(* Logix 5000 project; controller SX_V040001_C001 vendor 1 type 14 code 77 rev 16.23; software revision 16.04; part 20 of 35 *)
(* tags used below, declared in another part *)
   ALL_KINDS : INT[90];
   G_DInput : DINT[3];
   G_DOutput : DINT[3];
   METERING : INT[44];
   NOTDOS : INT[6];
   PARAMETER : INT[501];
(* MainProgram, continued *)

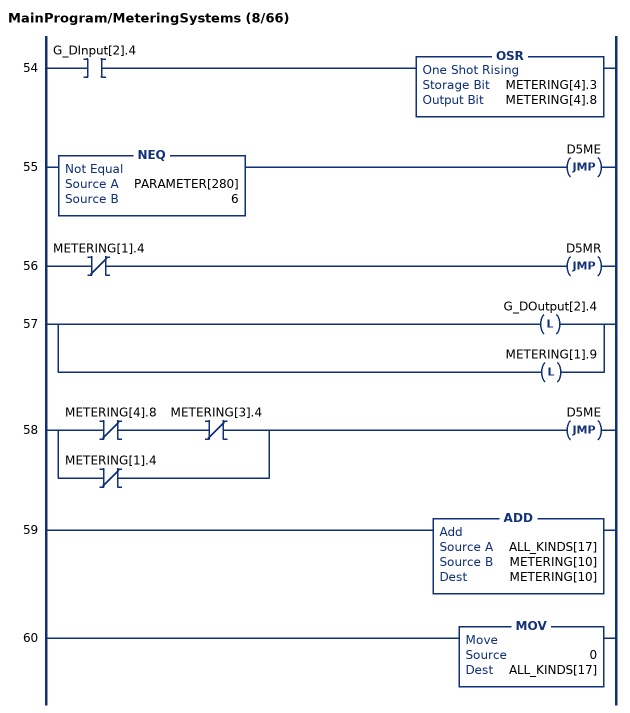
   [picture p432: MainProgram/MeteringSystems rungs 54-60]
   54: XIC(G_DInput[2].4)OSR(METERING[4].3,METERING[4].8);
   55: NEQ(PARAMETER[280],6)JMP(D5ME);
   56: XIO(METERING[1].4)JMP(D5MR);
   57: [OTL(G_DOutput[2].4) ,OTL(METERING[1].9) ];
   58: [XIO(METERING[4].8) XIO(METERING[3].4) ,XIO(METERING[1].4) ]JMP(D5ME);
   59: ADD(ALL_KINDS[17],METERING[10],METERING[10]);
   60: MOV(0,ALL_KINDS[17]);
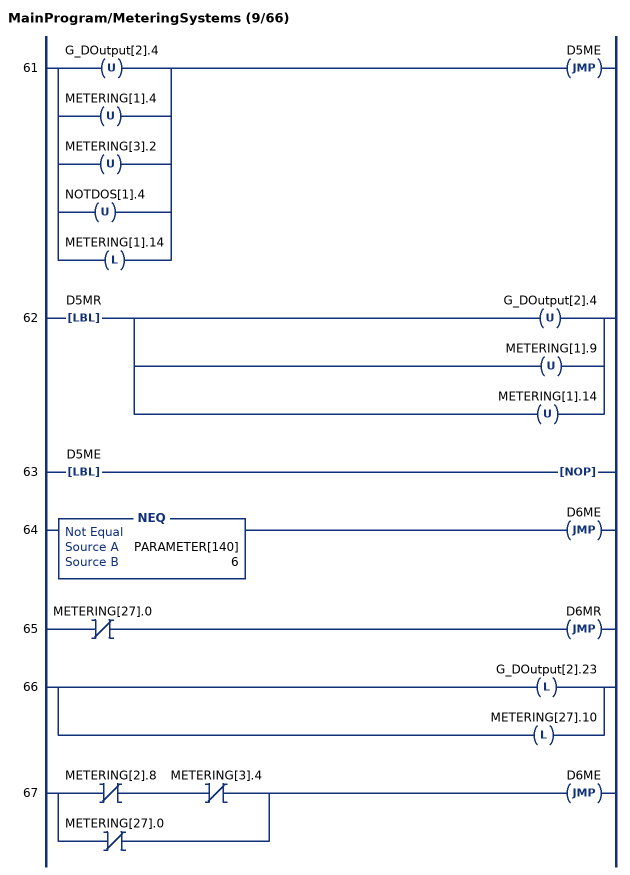
   61: [OTU(G_DOutput[2].4) ,OTU(METERING[1].4) ,OTU(METERING[3].2) ,OTU(NOTDOS[1].4) ,OTL(METERING[1].14) ]JMP(D5ME);
   62: LBL(D5MR)[OTU(G_DOutput[2].4) ,OTU(METERING[1].9) ,OTU(METERING[1].14) ];
   63: LBL(D5ME)NOP();
   64: NEQ(PARAMETER[140],6)JMP(D6ME);
   65: XIO(METERING[27].0)JMP(D6MR);
   66: [OTL(G_DOutput[2].23) ,OTL(METERING[27].10) ];
   67: [XIO(METERING[2].8) XIO(METERING[3].4) ,XIO(METERING[27].0) ]JMP(D6ME);
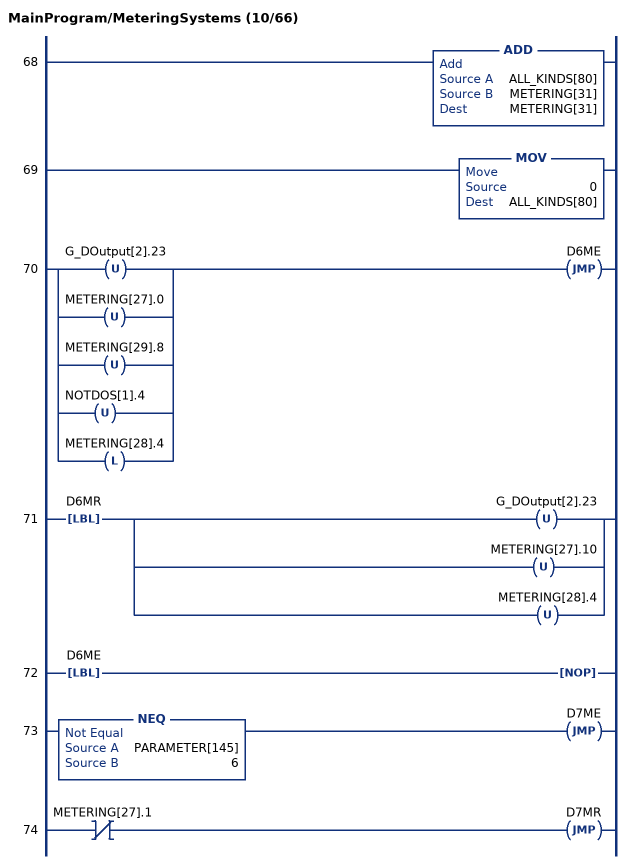
   68: ADD(ALL_KINDS[80],METERING[31],METERING[31]);
   69: MOV(0,ALL_KINDS[80]);
   70: [OTU(G_DOutput[2].23) ,OTU(METERING[27].0) ,OTU(METERING[29].8) ,OTU(NOTDOS[1].4) ,OTL(METERING[28].4) ]JMP(D6ME);
   71: LBL(D6MR)[OTU(G_DOutput[2].23) ,OTU(METERING[27].10) ,OTU(METERING[28].4) ];
   72: LBL(D6ME)NOP();
   73: NEQ(PARAMETER[145],6)JMP(D7ME);
   74: XIO(METERING[27].1)JMP(D7MR);
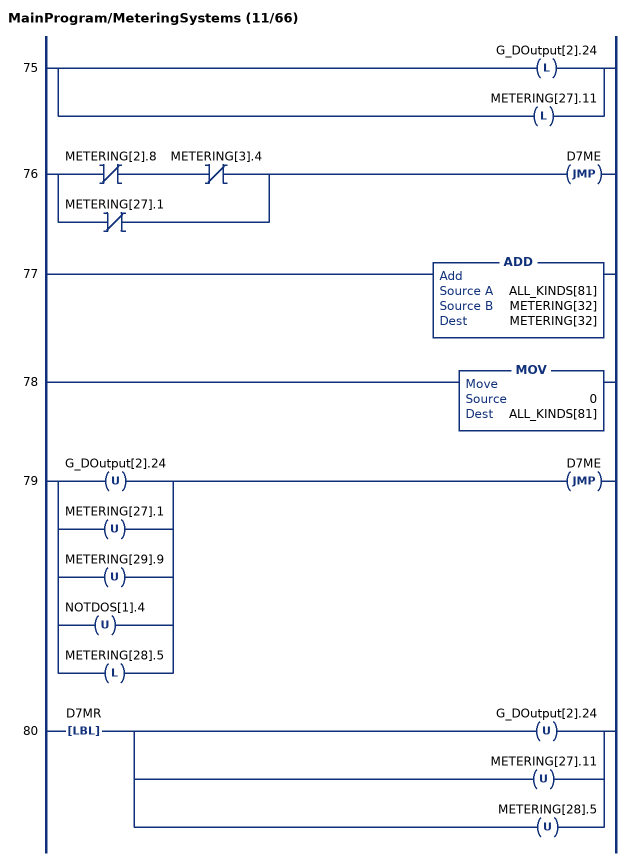
   75: [OTL(G_DOutput[2].24) ,OTL(METERING[27].11) ];
   76: [XIO(METERING[2].8) XIO(METERING[3].4) ,XIO(METERING[27].1) ]JMP(D7ME);
   77: ADD(ALL_KINDS[81],METERING[32],METERING[32]);
   78: MOV(0,ALL_KINDS[81]);
   79: [OTU(G_DOutput[2].24) ,OTU(METERING[27].1) ,OTU(METERING[29].9) ,OTU(NOTDOS[1].4) ,OTL(METERING[28].5) ]JMP(D7ME);
   80: LBL(D7MR)[OTU(G_DOutput[2].24) ,OTU(METERING[27].11) ,OTU(METERING[28].5) ];
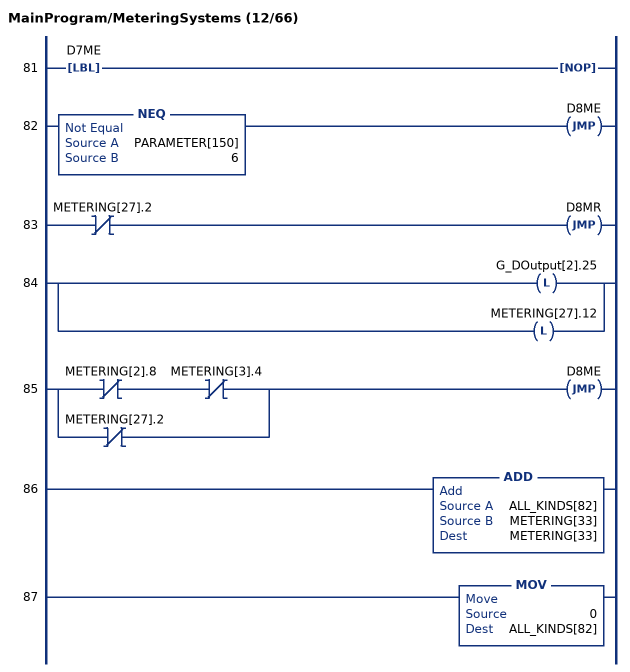
   81: LBL(D7ME)NOP();
   82: NEQ(PARAMETER[150],6)JMP(D8ME);
   83: XIO(METERING[27].2)JMP(D8MR);
   84: [OTL(G_DOutput[2].25) ,OTL(METERING[27].12) ];
   85: [XIO(METERING[2].8) XIO(METERING[3].4) ,XIO(METERING[27].2) ]JMP(D8ME);
   86: ADD(ALL_KINDS[82],METERING[33],METERING[33]);
   87: MOV(0,ALL_KINDS[82]);
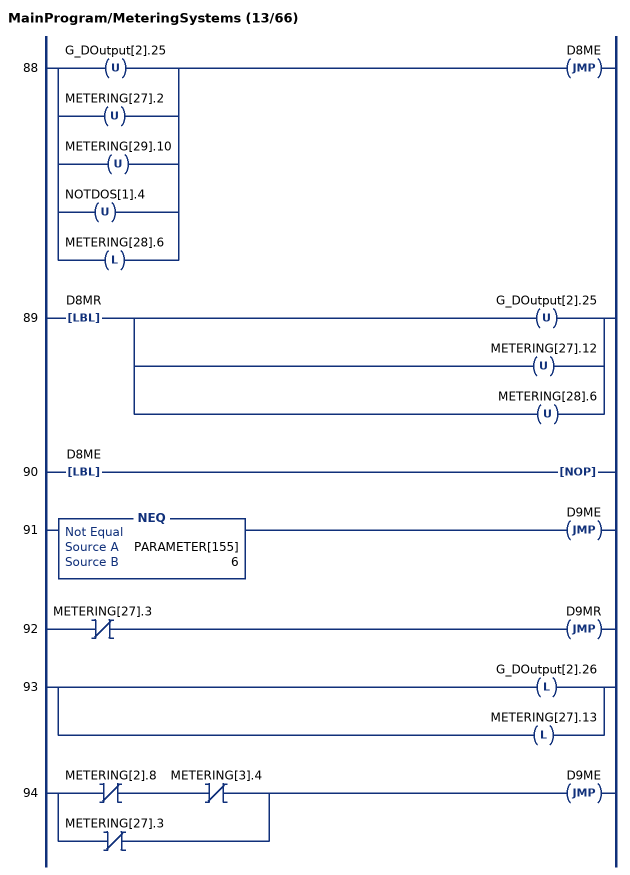
   88: [OTU(G_DOutput[2].25) ,OTU(METERING[27].2) ,OTU(METERING[29].10) ,OTU(NOTDOS[1].4) ,OTL(METERING[28].6) ]JMP(D8ME);
   89: LBL(D8MR)[OTU(G_DOutput[2].25) ,OTU(METERING[27].12) ,OTU(METERING[28].6) ];
   90: LBL(D8ME)NOP();
   91: NEQ(PARAMETER[155],6)JMP(D9ME);
   92: XIO(METERING[27].3)JMP(D9MR);
   93: [OTL(G_DOutput[2].26) ,OTL(METERING[27].13) ];
   94: [XIO(METERING[2].8) XIO(METERING[3].4) ,XIO(METERING[27].3) ]JMP(D9ME);
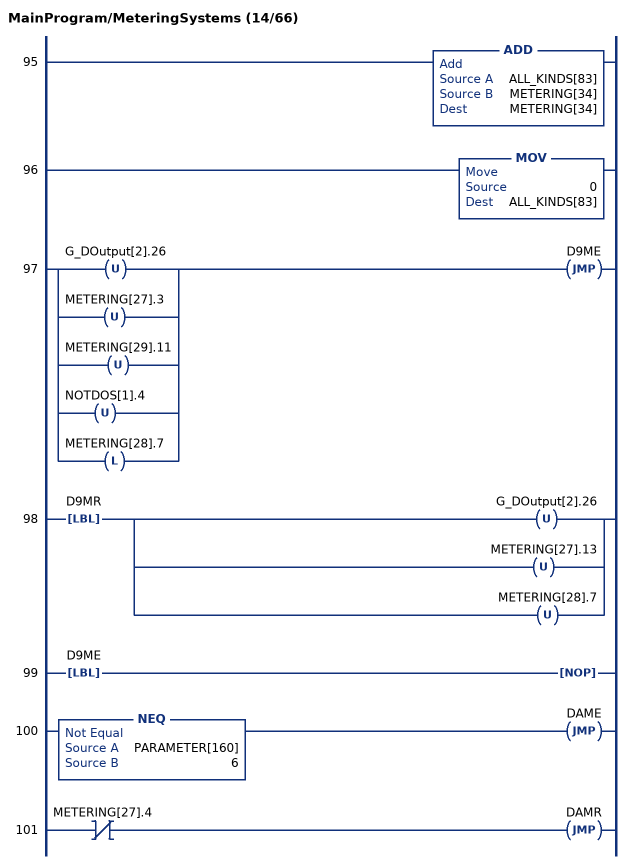
   95: ADD(ALL_KINDS[83],METERING[34],METERING[34]);
   96: MOV(0,ALL_KINDS[83]);
   97: [OTU(G_DOutput[2].26) ,OTU(METERING[27].3) ,OTU(METERING[29].11) ,OTU(NOTDOS[1].4) ,OTL(METERING[28].7) ]JMP(D9ME);
   98: LBL(D9MR)[OTU(G_DOutput[2].26) ,OTU(METERING[27].13) ,OTU(METERING[28].7) ];
   99: LBL(D9ME)NOP();
   100: NEQ(PARAMETER[160],6)JMP(DAME);
   101: XIO(METERING[27].4)JMP(DAMR);
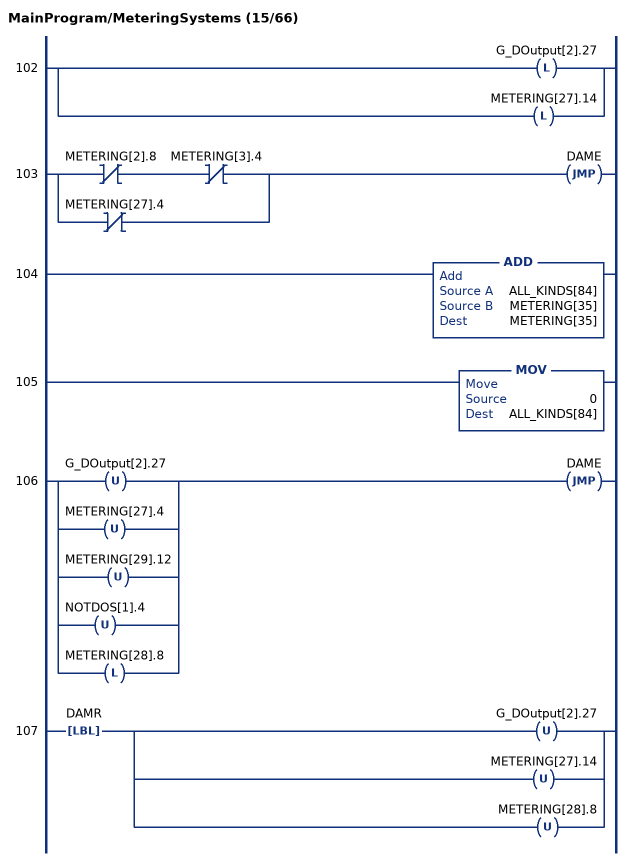
   102: [OTL(G_DOutput[2].27) ,OTL(METERING[27].14) ];
   103: [XIO(METERING[2].8) XIO(METERING[3].4) ,XIO(METERING[27].4) ]JMP(DAME);
   104: ADD(ALL_KINDS[84],METERING[35],METERING[35]);
   105: MOV(0,ALL_KINDS[84]);
   106: [OTU(G_DOutput[2].27) ,OTU(METERING[27].4) ,OTU(METERING[29].12) ,OTU(NOTDOS[1].4) ,OTL(METERING[28].8) ]JMP(DAME);
   107: LBL(DAMR)[OTU(G_DOutput[2].27) ,OTU(METERING[27].14) ,OTU(METERING[28].8) ];
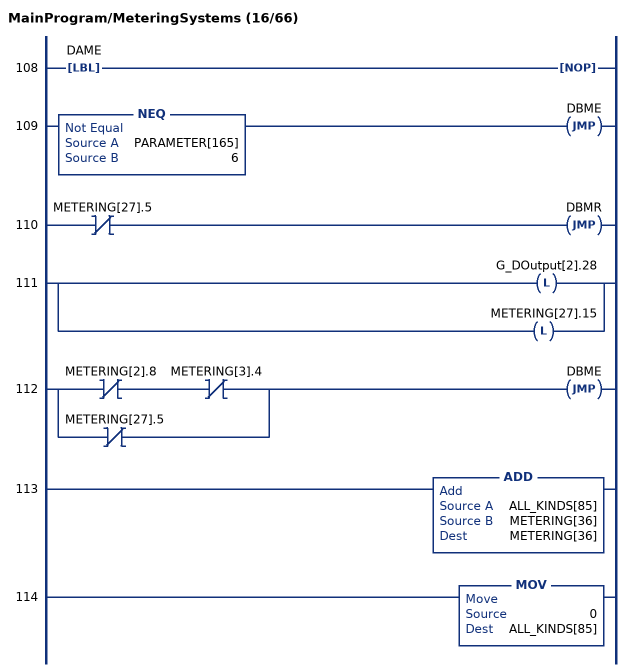
   108: LBL(DAME)NOP();
   109: NEQ(PARAMETER[165],6)JMP(DBME);
   110: XIO(METERING[27].5)JMP(DBMR);
   111: [OTL(G_DOutput[2].28) ,OTL(METERING[27].15) ];
   112: [XIO(METERING[2].8) XIO(METERING[3].4) ,XIO(METERING[27].5) ]JMP(DBME);
   113: ADD(ALL_KINDS[85],METERING[36],METERING[36]);
   114: MOV(0,ALL_KINDS[85]);
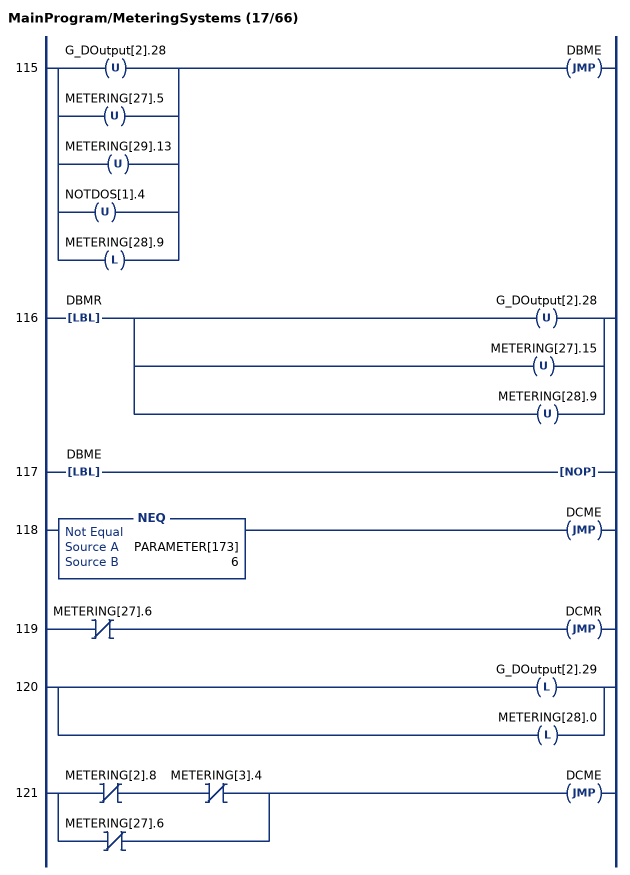
   115: [OTU(G_DOutput[2].28) ,OTU(METERING[27].5) ,OTU(METERING[29].13) ,OTU(NOTDOS[1].4) ,OTL(METERING[28].9) ]JMP(DBME);
   116: LBL(DBMR)[OTU(G_DOutput[2].28) ,OTU(METERING[27].15) ,OTU(METERING[28].9) ];
   117: LBL(DBME)NOP();
   118: NEQ(PARAMETER[173],6)JMP(DCME);
   119: XIO(METERING[27].6)JMP(DCMR);
   120: [OTL(G_DOutput[2].29) ,OTL(METERING[28].0) ];
   121: [XIO(METERING[2].8) XIO(METERING[3].4) ,XIO(METERING[27].6) ]JMP(DCME);
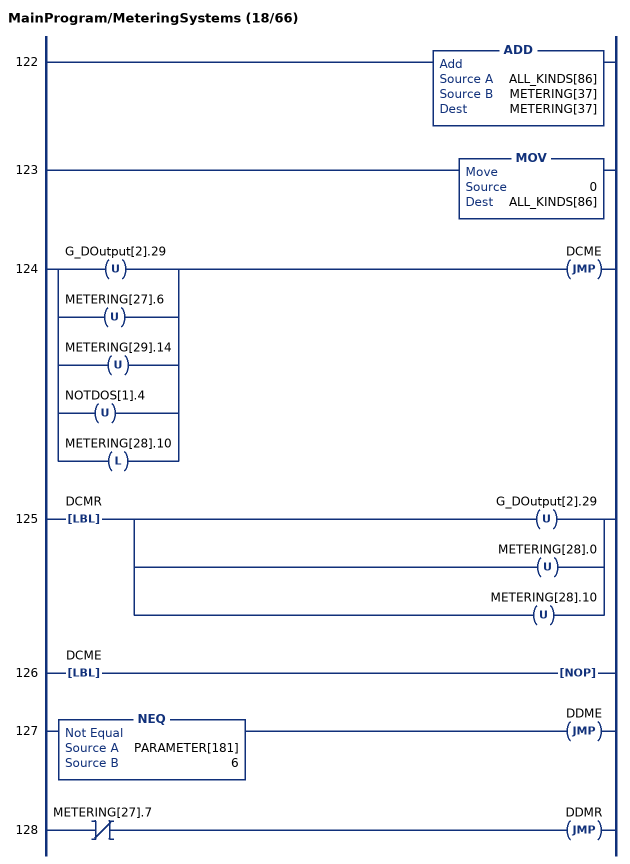
   122: ADD(ALL_KINDS[86],METERING[37],METERING[37]);
   123: MOV(0,ALL_KINDS[86]);
   124: [OTU(G_DOutput[2].29) ,OTU(METERING[27].6) ,OTU(METERING[29].14) ,OTU(NOTDOS[1].4) ,OTL(METERING[28].10) ]JMP(DCME);
   125: LBL(DCMR)[OTU(G_DOutput[2].29) ,OTU(METERING[28].0) ,OTU(METERING[28].10) ];
   126: LBL(DCME)NOP();
   127: NEQ(PARAMETER[181],6)JMP(DDME);
   128: XIO(METERING[27].7)JMP(DDMR);
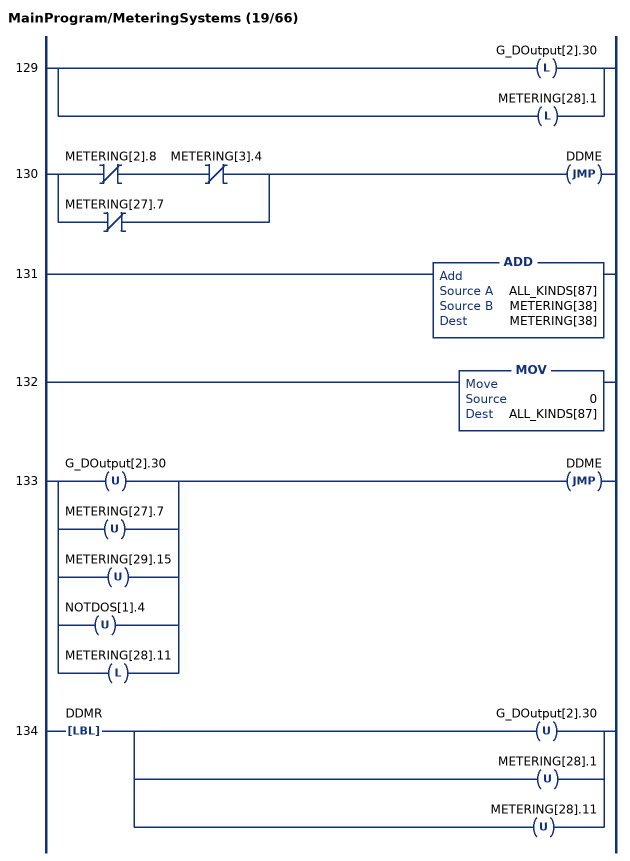
   129: [OTL(G_DOutput[2].30) ,OTL(METERING[28].1) ];
   130: [XIO(METERING[2].8) XIO(METERING[3].4) ,XIO(METERING[27].7) ]JMP(DDME);
   131: ADD(ALL_KINDS[87],METERING[38],METERING[38]);
   132: MOV(0,ALL_KINDS[87]);
   133: [OTU(G_DOutput[2].30) ,OTU(METERING[27].7) ,OTU(METERING[29].15) ,OTU(NOTDOS[1].4) ,OTL(METERING[28].11) ]JMP(DDME);
   134: LBL(DDMR)[OTU(G_DOutput[2].30) ,OTU(METERING[28].1) ,OTU(METERING[28].11) ];
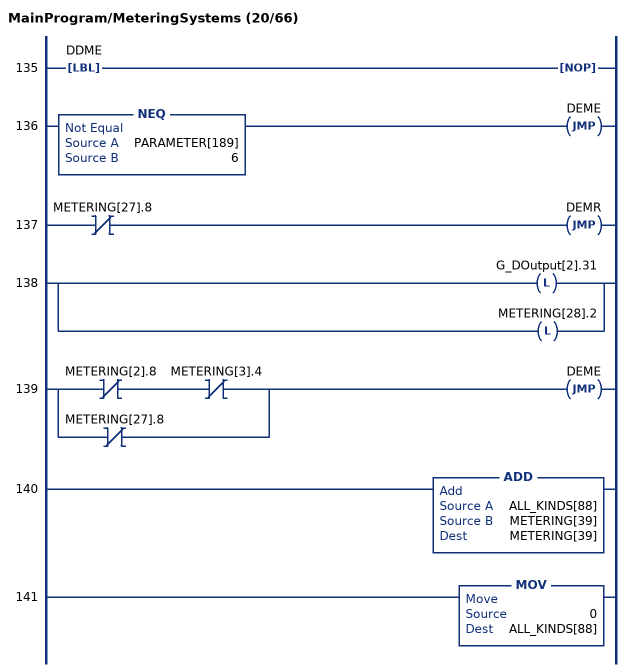
   135: LBL(DDME)NOP();
   136: NEQ(PARAMETER[189],6)JMP(DEME);
   137: XIO(METERING[27].8)JMP(DEMR);
   138: [OTL(G_DOutput[2].31) ,OTL(METERING[28].2) ];
   139: [XIO(METERING[2].8) XIO(METERING[3].4) ,XIO(METERING[27].8) ]JMP(DEME);
   140: ADD(ALL_KINDS[88],METERING[39],METERING[39]);
   141: MOV(0,ALL_KINDS[88]);
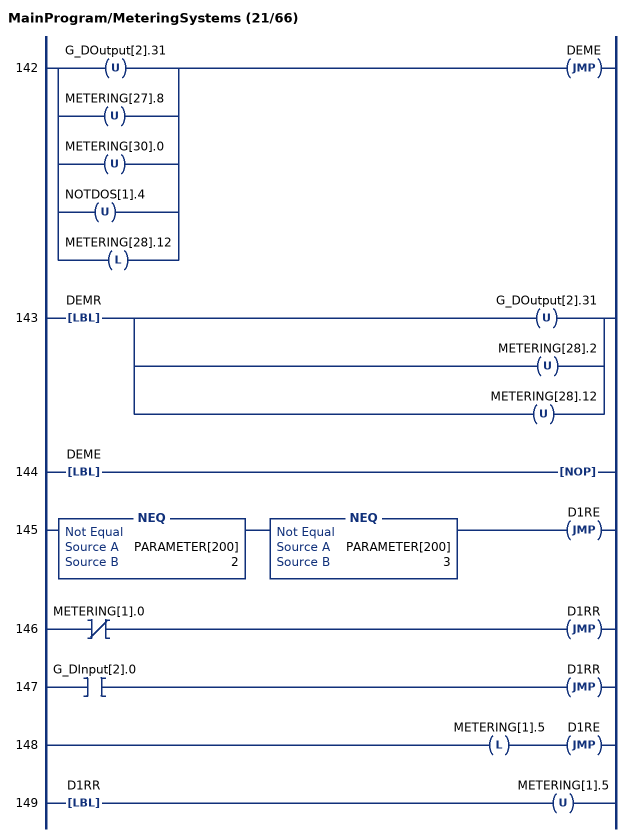
   142: [OTU(G_DOutput[2].31) ,OTU(METERING[27].8) ,OTU(METERING[30].0) ,OTU(NOTDOS[1].4) ,OTL(METERING[28].12) ]JMP(DEME);
   143: LBL(DEMR)[OTU(G_DOutput[2].31) ,OTU(METERING[28].2) ,OTU(METERING[28].12) ];
   144: LBL(DEME)NOP();
   145: NEQ(PARAMETER[200],2)NEQ(PARAMETER[200],3)JMP(D1RE);
   146: XIO(METERING[1].0)JMP(D1RR);
   147: XIC(G_DInput[2].0)JMP(D1RR);
   148: OTL(METERING[1].5)JMP(D1RE);
   149: LBL(D1RR)OTU(METERING[1].5);
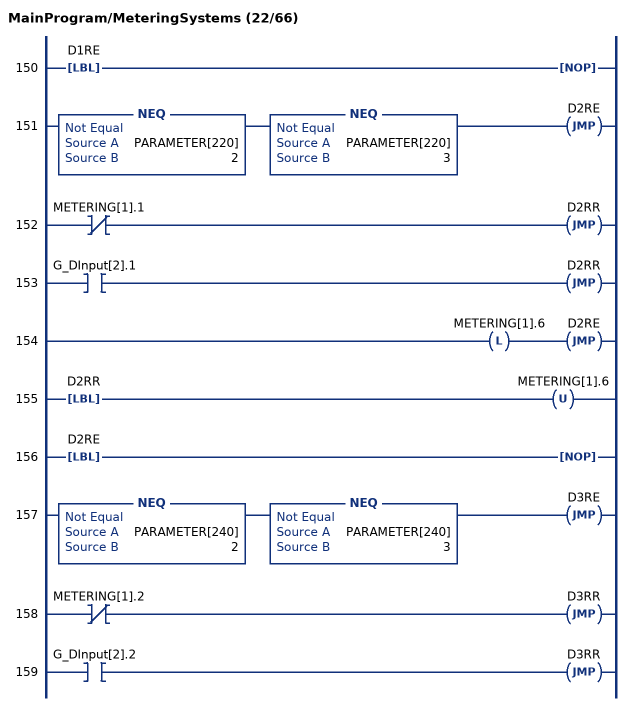
   150: LBL(D1RE)NOP();
   151: NEQ(PARAMETER[220],2)NEQ(PARAMETER[220],3)JMP(D2RE);
   152: XIO(METERING[1].1)JMP(D2RR);
   153: XIC(G_DInput[2].1)JMP(D2RR);
   154: OTL(METERING[1].6)JMP(D2RE);
   155: LBL(D2RR)OTU(METERING[1].6);
   156: LBL(D2RE)NOP();
   157: NEQ(PARAMETER[240],2)NEQ(PARAMETER[240],3)JMP(D3RE);
   158: XIO(METERING[1].2)JMP(D3RR);
   159: XIC(G_DInput[2].2)JMP(D3RR);
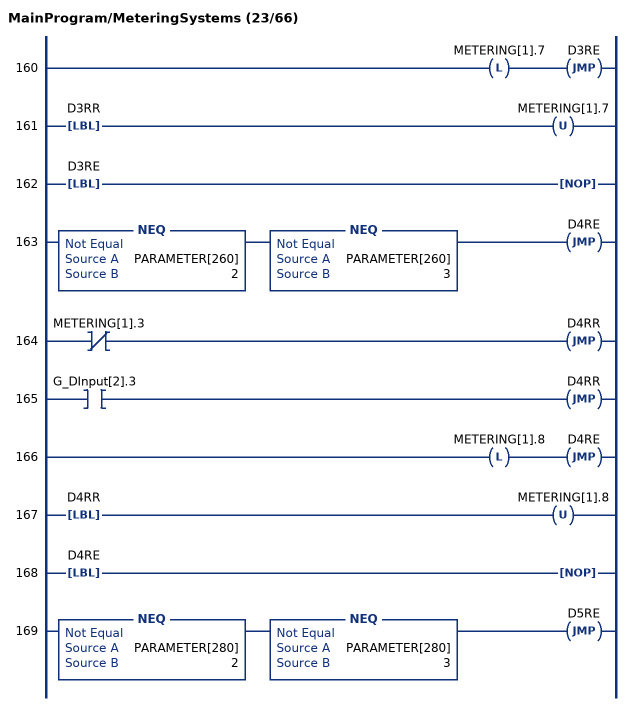
   160: OTL(METERING[1].7)JMP(D3RE);
   161: LBL(D3RR)OTU(METERING[1].7);
   162: LBL(D3RE)NOP();
   163: NEQ(PARAMETER[260],2)NEQ(PARAMETER[260],3)JMP(D4RE);
   164: XIO(METERING[1].3)JMP(D4RR);
   165: XIC(G_DInput[2].3)JMP(D4RR);
   166: OTL(METERING[1].8)JMP(D4RE);
   167: LBL(D4RR)OTU(METERING[1].8);
   168: LBL(D4RE)NOP();
   169: NEQ(PARAMETER[280],2)NEQ(PARAMETER[280],3)JMP(D5RE);
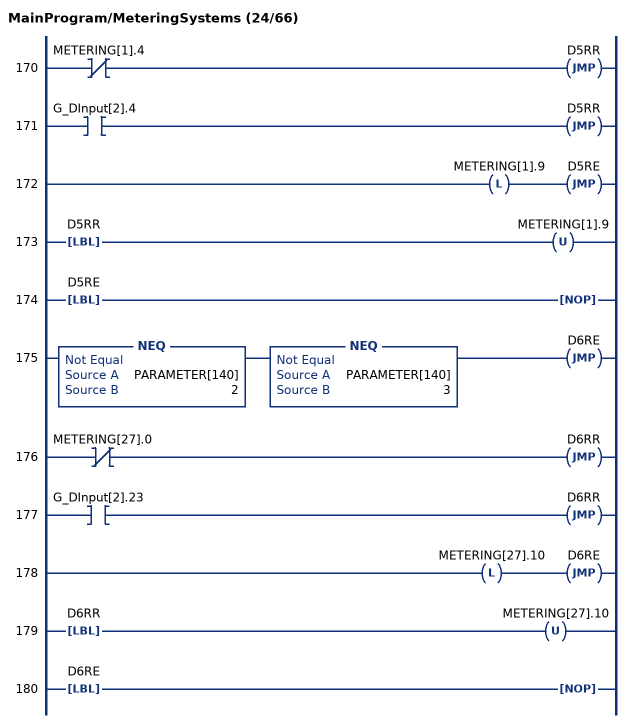
   170: XIO(METERING[1].4)JMP(D5RR);
   171: XIC(G_DInput[2].4)JMP(D5RR);
   172: OTL(METERING[1].9)JMP(D5RE);
   173: LBL(D5RR)OTU(METERING[1].9);
   174: LBL(D5RE)NOP();
   175: NEQ(PARAMETER[140],2)NEQ(PARAMETER[140],3)JMP(D6RE);
   176: XIO(METERING[27].0)JMP(D6RR);
   177: XIC(G_DInput[2].23)JMP(D6RR);
   178: OTL(METERING[27].10)JMP(D6RE);
   179: LBL(D6RR)OTU(METERING[27].10);
   180: LBL(D6RE)NOP();
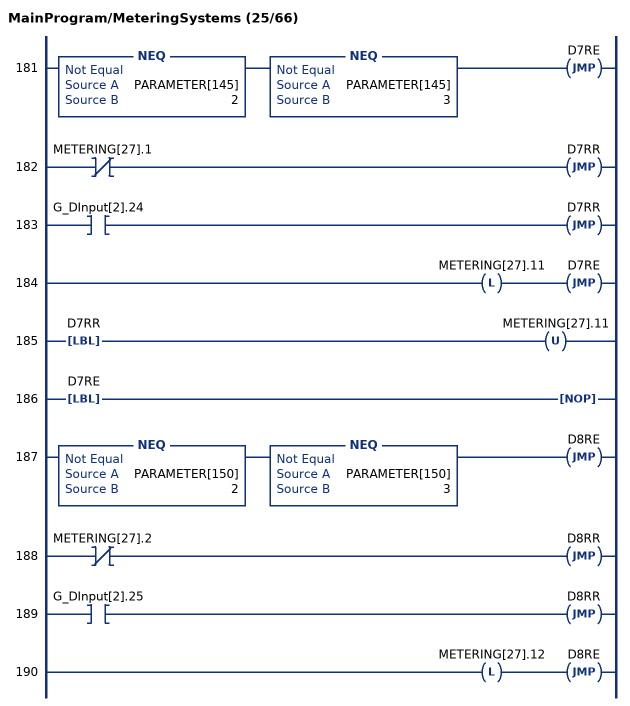
   181: NEQ(PARAMETER[145],2)NEQ(PARAMETER[145],3)JMP(D7RE);
   182: XIO(METERING[27].1)JMP(D7RR);
   183: XIC(G_DInput[2].24)JMP(D7RR);
   184: OTL(METERING[27].11)JMP(D7RE);
   185: LBL(D7RR)OTU(METERING[27].11);
   186: LBL(D7RE)NOP();
   187: NEQ(PARAMETER[150],2)NEQ(PARAMETER[150],3)JMP(D8RE);
   188: XIO(METERING[27].2)JMP(D8RR);
   189: XIC(G_DInput[2].25)JMP(D8RR);
   190: OTL(METERING[27].12)JMP(D8RE);
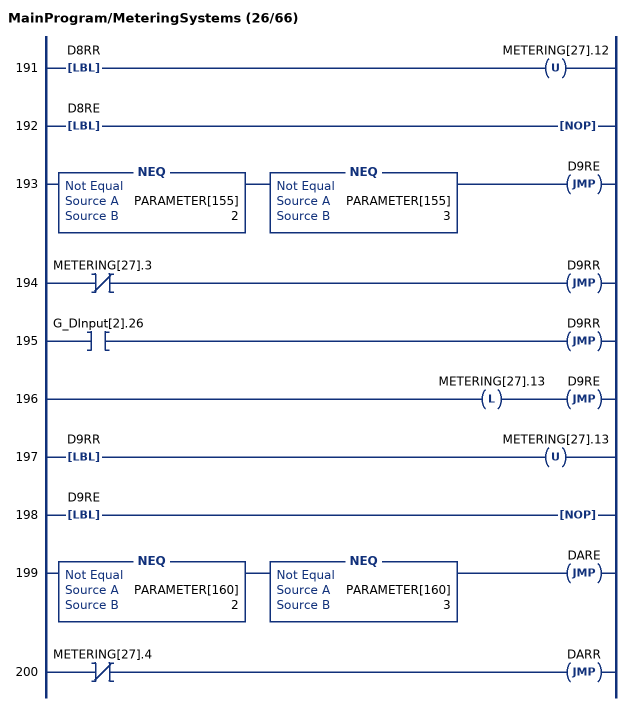
   191: LBL(D8RR)OTU(METERING[27].12);
   192: LBL(D8RE)NOP();
   193: NEQ(PARAMETER[155],2)NEQ(PARAMETER[155],3)JMP(D9RE);
   194: XIO(METERING[27].3)JMP(D9RR);
   195: XIC(G_DInput[2].26)JMP(D9RR);
   196: OTL(METERING[27].13)JMP(D9RE);
   197: LBL(D9RR)OTU(METERING[27].13);
   198: LBL(D9RE)NOP();
   199: NEQ(PARAMETER[160],2)NEQ(PARAMETER[160],3)JMP(DARE);
   200: XIO(METERING[27].4)JMP(DARR);
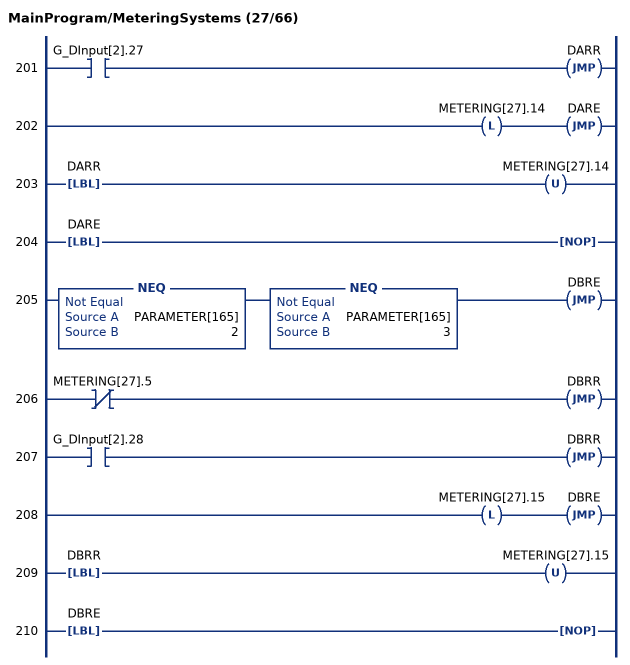
   201: XIC(G_DInput[2].27)JMP(DARR);
   202: OTL(METERING[27].14)JMP(DARE);
   203: LBL(DARR)OTU(METERING[27].14);
   204: LBL(DARE)NOP();
   205: NEQ(PARAMETER[165],2)NEQ(PARAMETER[165],3)JMP(DBRE);
   206: XIO(METERING[27].5)JMP(DBRR);
   207: XIC(G_DInput[2].28)JMP(DBRR);
   208: OTL(METERING[27].15)JMP(DBRE);
   209: LBL(DBRR)OTU(METERING[27].15);
   210: LBL(DBRE)NOP();
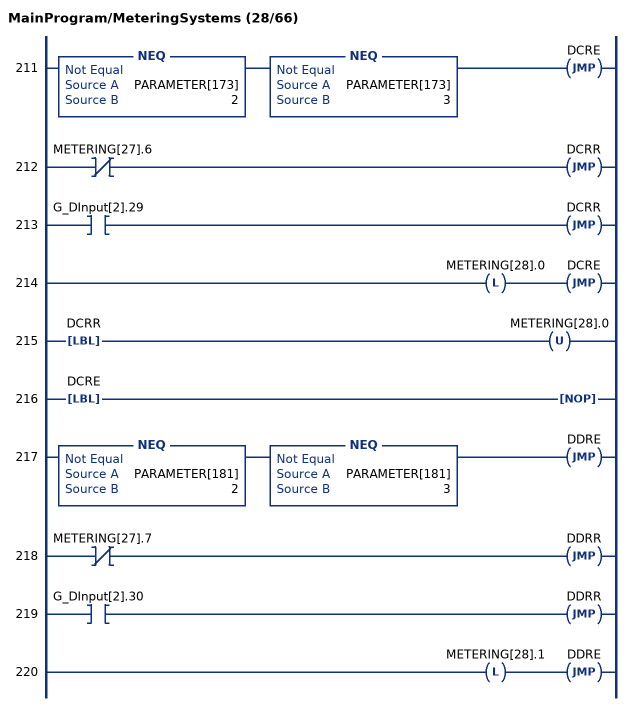
   211: NEQ(PARAMETER[173],2)NEQ(PARAMETER[173],3)JMP(DCRE);
   212: XIO(METERING[27].6)JMP(DCRR);
   213: XIC(G_DInput[2].29)JMP(DCRR);
   214: OTL(METERING[28].0)JMP(DCRE);
   215: LBL(DCRR)OTU(METERING[28].0);
   216: LBL(DCRE)NOP();
   217: NEQ(PARAMETER[181],2)NEQ(PARAMETER[181],3)JMP(DDRE);
   218: XIO(METERING[27].7)JMP(DDRR);
   219: XIC(G_DInput[2].30)JMP(DDRR);
   220: OTL(METERING[28].1)JMP(DDRE);
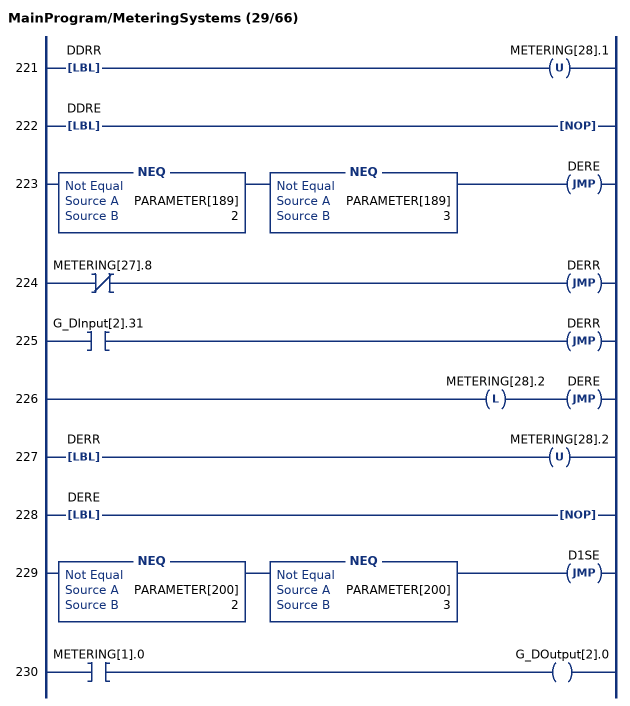
   221: LBL(DDRR)OTU(METERING[28].1);
   222: LBL(DDRE)NOP();
   223: NEQ(PARAMETER[189],2)NEQ(PARAMETER[189],3)JMP(DERE);
   224: XIO(METERING[27].8)JMP(DERR);
   225: XIC(G_DInput[2].31)JMP(DERR);
   226: OTL(METERING[28].2)JMP(DERE);
   227: LBL(DERR)OTU(METERING[28].2);
   228: LBL(DERE)NOP();
   229: NEQ(PARAMETER[200],2)NEQ(PARAMETER[200],3)JMP(D1SE);
   230: XIC(METERING[1].0)OTE(G_DOutput[2].0);
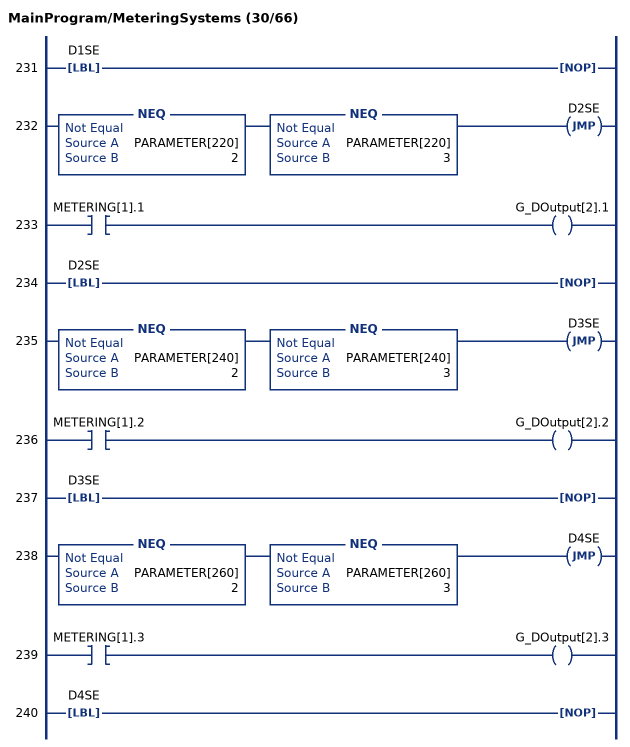
   231: LBL(D1SE)NOP();
   232: NEQ(PARAMETER[220],2)NEQ(PARAMETER[220],3)JMP(D2SE);
   233: XIC(METERING[1].1)OTE(G_DOutput[2].1);
   234: LBL(D2SE)NOP();
   235: NEQ(PARAMETER[240],2)NEQ(PARAMETER[240],3)JMP(D3SE);
   236: XIC(METERING[1].2)OTE(G_DOutput[2].2);
   237: LBL(D3SE)NOP();
   238: NEQ(PARAMETER[260],2)NEQ(PARAMETER[260],3)JMP(D4SE);
   239: XIC(METERING[1].3)OTE(G_DOutput[2].3);
   240: LBL(D4SE)NOP();
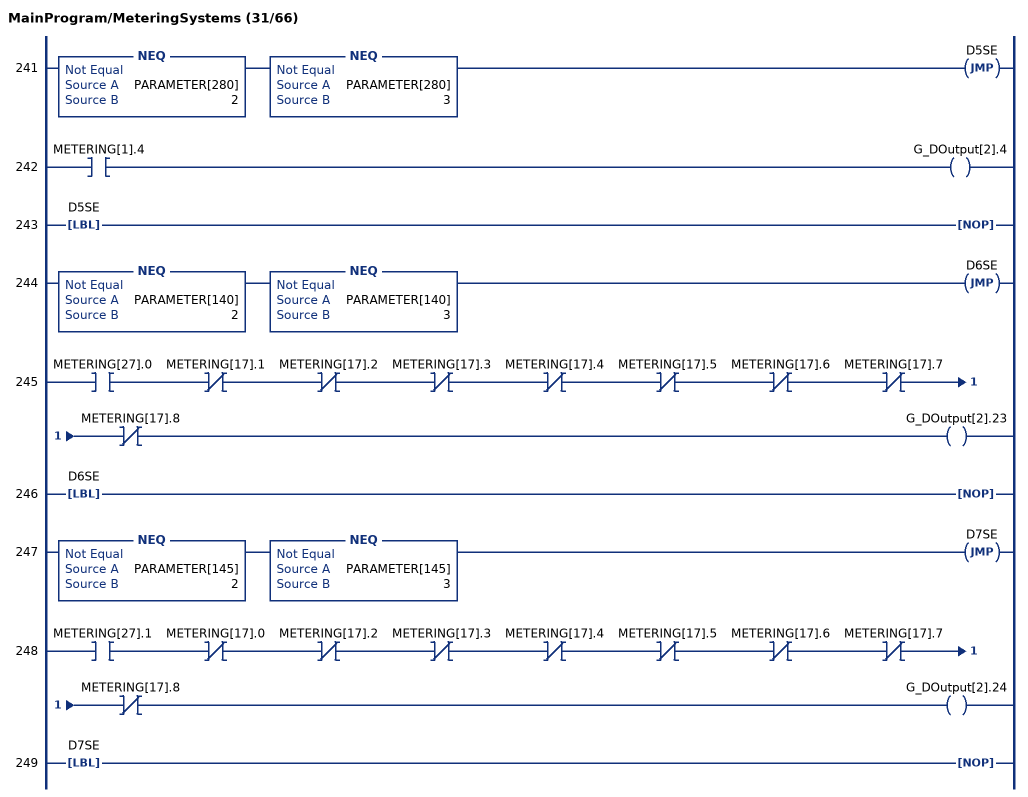
   241: NEQ(PARAMETER[280],2)NEQ(PARAMETER[280],3)JMP(D5SE);
   242: XIC(METERING[1].4)OTE(G_DOutput[2].4);
   243: LBL(D5SE)NOP();
   244: NEQ(PARAMETER[140],2)NEQ(PARAMETER[140],3)JMP(D6SE);
   245: XIC(METERING[27].0)XIO(METERING[17].1)XIO(METERING[17].2)XIO(METERING[17].3)XIO(METERING[17].4)XIO(METERING[17].5)XIO(METERING[17].6)XIO(METERING[17].7)XIO(METERING[17].8)OTE(G_DOutput[2].23);
   246: LBL(D6SE)NOP();
   247: NEQ(PARAMETER[145],2)NEQ(PARAMETER[145],3)JMP(D7SE);
   248: XIC(METERING[27].1)XIO(METERING[17].0)XIO(METERING[17].2)XIO(METERING[17].3)XIO(METERING[17].4)XIO(METERING[17].5)XIO(METERING[17].6)XIO(METERING[17].7)XIO(METERING[17].8)OTE(G_DOutput[2].24);
   249: LBL(D7SE)NOP();
